PROGRAM RECIPE_Controller
VAR	
END_VAR

END_PROGRAM

(* stored: Version 1.1.0.1, ProductVersion 3.1.4022.18
   POU RECIPE_Controller: Id {fe0b8a2c-7755-48b6-8b7f-aa457ab7aa7b}, SpecialFunc None *)
